(* CODESYS project IndraLogic.project

Project tree, tasks and I/O mapping:
  Sortierstrecke_SPS : IndraControl XM2, Bosch Rexroth AG, order no. dependent on customer specific configuration, version 14.20.34.0
    application Application
      libraries: CommonDataTypes, 3.5.8.40 (OSB AG)
      task PlcTask (cyclic, interval 10 ms, priority 5, watchdog 10 ms x 2) calls PlcProg
      controller/
        function block ColorSensor [ST]: toInt
        function block Compressor [ST]: isActive, start, stop
        function block Conveyor [ST]: isActive, start, stop
        function block Cylinder [ST]: isHome, isWork, moveHome, moveWork
      GVL/
        global variables GVL_IO
        global variables GVL_MasterSlave
        global variables NVL_I_Sorter
        declarations NVL_O_Sorter
      SPS_Communication/
        function block ReadOutputs [ST]: get
        function block SendInputs [ST]: set
      global variables UserVarGlobal
      function CheckBounds [ST]
      program PlcProg [ST]
      program PlcStudentProg [ST]
      Symbols
      visualisation Visualization
    S20_I_O : S20_I_O, Bosch Rexroth AG, version 14.20.10.0
      S20_DIDO_8_1 : S20-DIDO-8/1, Bosch Rexroth AG, order no. R911173745, version Revision=16#0
          settings: Digital Input.IDN = 16#010005DF; Digital Output.IDN = 16#010005DE; Digital Input.IDN = 16#010005DF; Digital Input.Process data out.IDN = 16#00000000; Digital Input.Process data in.IDN = 16#010905DF; Digital Input.Diag out.IDN = 16#00000000; Digital Input.Diag in.IDN = 16#00000000; Digital Input.Io monitoring.IDN_IN = 16#00000000; Digital Input.Io monitoring.IDN_OUT = 16#00000000; Digital Output.IDN = 16#010005DE; Digital Output.Process data out.IDN = 16#010505DE; Digital Output.Process data in.IDN = 16#00000000; Digital Output.Diag out.IDN = 16#00000000; Digital Output.Diag in.IDN = 16#00000000; Digital Output.Io monitoring.IDN_IN = 16#00000000; Digital Output.Io monitoring.IDN_OUT = 16#00000000; PropritaryParameterSet_S-0-1503.0.20.IDN = 16#011405DF; PropritaryParameterSet_S-0-1502.0.2.IDN = 16#010205DE
          output Application.GVL_IO.DO_MotorBeltForward : BOOL  // Digital Output.02
          output Application.GVL_IO.DO_Compressor : BOOL  // Digital Output.03
          output Application.GVL_IO.DO_ValceEjectorOne : BOOL  // Digital Output.12
          output Application.GVL_IO.DO_ValceEjectorTwo : BOOL  // Digital Output.13
          output Application.GVL_IO.DO_ValceEjectorThree : BOOL  // Digital Output.22
          input  Application.GVL_IO.DI_LightBarrierInlet : BOOL  // Digital Input.00
          input  Application.GVL_IO.DI_LightBarrierBehindColor : BOOL  // Digital Input.01
          input  Application.GVL_IO.DI_LightBarrierWhite : BOOL  // Digital Input.10
          input  Application.GVL_IO.DI_LightBarrierRed : BOOL  // Digital Input.11
          input  Application.GVL_IO.DI_LightBarrierBlue : BOOL  // Digital Input.20
          input  Application.GVL_IO.DI_PulseCounter : BOOL  // Digital Input.21
          unmapped channels: Digital Output, Digital Input
      S20_AI_4_U : S20-AI-4-U, Bosch Rexroth AG, order no. R911173256, version Revision=16#0
          settings: Analog Input.IDN = 16#010005E1; Analog Input.IDN = 16#010005E1; Analog Input.Process data out.IDN = 16#00000000; Analog Input.Process data in.IDN = 16#010905E1; Analog Input.Diag out.IDN = 16#00000000; Analog Input.Diag in.IDN = 16#00000000; Analog Input.Io monitoring.IDN_IN = 16#00000000; Analog Input.Io monitoring.IDN_OUT = 16#00000000; PropritaryParameterSet_P-1-0128.0.0.IDN = 16#01009080; PropritaryParameterSet_P-1-0128.0.0.Abort if error = False; PropritaryParameterSet_P-1-0128.0.0.Jump to line if error = False; PropritaryParameterSet_P-1-0128.0.0.SercosAttribute = 16#00000000; PropritaryParameterSet_P-1-0128.0.0 = [16#0C,16#00,16#0C,16#00,16#00,16#02,16#00,16#0F,16#00,16#0F,16#00,16#0F,16#00,16#00,16#00,16#00]
          input  Application.GVL_IO.AI_ColorSensor : WORD  // Analog Input.Analog Input 1
          unmapped channels: Analog Input
    Nicht_verwendet_XM_ : Nicht verwendet (XM), Bosch Rexroth AG, version 14.18.0.0
  text list GlobalTextList
*)

// Sortierstrecke_SPS/Application/GVL/GVL_IO
{attribute 'qualified_only'}
VAR_GLOBAL
		
	//Motors
	DO_MotorBeltForward				: BOOL; //Q1 AT	%QX0.0 
	//Pipes
	DO_Compressor					: BOOL; //Q2 AT	%QX0.1 
	DO_ValceEjectorOne				: BOOL; //Q3 AT	%QX0.2 
	DO_ValceEjectorTwo				: BOOL; //Q4 AT	%QX0.3 
	DO_ValceEjectorThree			: BOOL; //Q5 AT	%QX0.4 
	
	//Pulse Counter
	DI_PulseCounter				 	: BOOL; //I1 AT 	%IX0.5 
	//Light Barriers
	DI_LightBarrierInlet			: BOOL; //I2 AT 	%IX0.0 
	DI_LightBarrierBehindColor 		: BOOL; //I3 AT 	%IX0.1 
	DI_LightBarrierWhite			: BOOL; //I5 AT 	%IX0.2 
	DI_LightBarrierRed	 			: BOOL; //I6 AT 	%IX0.3 
	DI_LightBarrierBlue		 		: BOOL; //I7 AT 	%IX0.4 

	//Color Sensor
	AI_ColorSensor					: WORD; //A4 AT 	%IW2   	
END_VAR

// Sortierstrecke_SPS/Application/GVL/GVL_MasterSlave
{attribute 'qualified_only'}
VAR_GLOBAL
	runMaster : BOOL;
	Stop : BOOL;
END_VAR

// Sortierstrecke_SPS/Application/GVL/NVL_I_Sorter
{attribute 'qualified_only'}
VAR_GLOBAL
	
	//
	//INPUTS:
	//
	
	//Pulse Counter
	DI_PulseCounter				 	: BOOL; //I1 AT 	%IX0.5 
	//Light Barriers
	DI_LightBarrierInlet			: BOOL; //I2 AT 	%IX0.0 
	DI_LightBarrierBehindColor 		: BOOL; //I3 AT 	%IX0.1 
	DI_LightBarrierWhite			: BOOL; //I5 AT 	%IX0.2 
	DI_LightBarrierRed	 			: BOOL; //I6 AT 	%IX0.3 
	DI_LightBarrierBlue		 		: BOOL; //I7 AT 	%IX0.4 

	//Color Sensor
	AI_ColorSensor					: WORD; //A4 AT 	%IW2   	

END_VAR

// Sortierstrecke_SPS/Application/GVL/NVL_O_Sorter
//Diese globale Variablenliste wird über das Netzwerk empfangen.
//Sender: Import aus Datei 'C:\Users\tdie\Documents\HTWK_einzeln\Final\GVLs\Sorter_O.gvl'
//Protokoll: UDP

{attribute 'qualified_only'}
VAR_GLOBAL
	//
	//OUTPUTS:
	//
	
	//Motors
	DO_MotorBeltForward				: BOOL; //Q1 AT	%QX0.0 
	//Pipes
	DO_Compressor					: BOOL; //Q2 AT	%QX0.1 
	DO_ValceEjectorOne				: BOOL; //Q3 AT	%QX0.2 
	DO_ValceEjectorTwo				: BOOL; //Q4 AT	%QX0.3 
	DO_ValceEjectorThree			: BOOL; //Q5 AT	%QX0.4 
	
	Stop : BOOL;
	
END_VAR

// Sortierstrecke_SPS/Application/UserVarGlobal
{attribute 'qualified_only'}
VAR_GLOBAL
	// speichert die Farbe als INT - Wert
	colorAsInt 		: INT;
	
	//zählt die steigenden Flanken des Puls - Counters, um die Position des Objektes
	// auf dem Band zu bestimmen
	clock 	: INT;
END_VAR

// Sortierstrecke_SPS/Application/PlcProg
PROGRAM PlcProg
VAR
	reader : ReadOutputs();
	writer : SendInputs();
END_VAR

//---------------------------------------------------------------
//|		-			run the student code				-		|			
//---------------------------------------------------------------
PlcStudentProg();

//---------------------------------------------------------------
//|		-		Communication, do not modify!			-		|			
//---------------------------------------------------------------

writer.set();
reader.get();

END_PROGRAM

// Sortierstrecke_SPS/Application/PlcStudentProg
PROGRAM PlcStudentProg
VAR
	ColorSensorController	: ColorSensor;
	CompressorController	: Compressor;
	ConveyorController		: Conveyor;
	CylinderController		: Cylinder;
END_VAR

//---------------------------------------------------------------
//|		-		activate or deactivate Master			-		|			
//---------------------------------------------------------------

GVL_MasterSlave.runMaster := FALSE;

//---------------------------------------------------------------
//|		-		write your own code here				-		|			
//---------------------------------------------------------------

ColorSensorController(
	LightValue 				:= GVL_IO.AI_ColorSensor,
	clock					:= UserVarGlobal.clock);
UserVarGlobal.colorAsInt 	:= ColorSensorController.colorAsInt;

CompressorController(
	LightBarrierInlet 		:= GVL_IO.DI_LightBarrierInlet,
	LightBarrierWhite 		:= GVL_IO.DI_LightBarrierWhite,
	LightBarrierBlue 		:= GVL_IO.DI_LightBarrierBlue, 
	LightBarrierRed 		:= GVL_IO.DI_LightBarrierRed);
GVL_IO.DO_Compressor 		:= CompressorController.CompressorM;

ConveyorController(
	LightBarrierWhite		:= GVL_IO.DI_LightBarrierWhite,
	LightBarrierRed			:= GVL_IO.DI_LightBarrierRed,
	LightBarrierBlue		:= GVL_IO.DI_LightBarrierBlue,
	LightBarrierInlet		:= GVL_IO.DI_LightBarrierInlet,
	PulseCounter			:= GVL_IO.DI_PulseCounter);
GVL_IO.DO_MotorBeltForward 	:= ConveyorController.MotorBeltForward;
UserVarGlobal.clock		 	:= ConveyorController.clock;

CylinderController(
	colorAsInt 				:= UserVarGlobal.colorAsInt,
	clock		 			:= UserVarGlobal.clock);
GVL_IO.DO_ValceEjectorOne 	:= CylinderController.ValceEjectorOne;
GVL_IO.DO_ValceEjectorTwo 	:= CylinderController.ValceEjectorTwo;
GVL_IO.DO_ValceEjectorThree := CylinderController.ValceEjectorThree;

END_PROGRAM

// Sortierstrecke_SPS/Application/controller/ColorSensor
FUNCTION_BLOCK ColorSensor
VAR_INPUT
	LightValue	: DWORD;
	clock		: INT;
END_VAR
VAR_OUTPUT
	colorAsInt	: INT;
END_VAR
VAR
	
END_VAR

IF clock = 1 THEN
	THIS^.colorAsInt := toInt();
END_IF

METHOD toInt : INT
VAR_INPUT
END_VAR
IF THIS^.LightValue = 0 THEN
	toInt := 0;	//white
ELSIF THIS^.LightValue = 1 THEN
	toInt := 1; //red
ELSIF THIS^.LightValue = 2 THEN
	toInt := 2; //blue
ELSE 
	toInt := 3; //sollte nicht passieren
END_IF;
END_METHOD

END_FUNCTION_BLOCK

// Sortierstrecke_SPS/Application/controller/Compressor
FUNCTION_BLOCK Compressor

VAR_INPUT
	LightBarrierInlet			: BOOL;
	LightBarrierWhite 		 	: BOOL;
	LightBarrierBlue 			: BOOL;
	LightBarrierRed 			: BOOL;
END_VAR
VAR_OUTPUT
	CompressorM					: BOOL;
END_VAR
VAR
	an : F_TRIG;
	aus : F_TRIG;
END_VAR

an(CLK := LightBarrierInlet);
aus(CLK := LightBarrierWhite AND  LightBarrierBlue AND LightBarrierRed);

//Laden
IF an.Q AND NOT isActive() THEN
	start();
END_IF

//Stoppen
IF aus.Q AND isActive() THEN
	stop();
END_IF

METHOD isActive : BOOL
VAR_INPUT
END_VAR
IF THIS^.CompressorM THEN
	isActive := TRUE;
ELSE
	isActive := FALSE;
END_IF
END_METHOD

METHOD start
VAR_INPUT
END_VAR
THIS^.CompressorM := TRUE;
END_METHOD

METHOD stop
VAR_INPUT
END_VAR
THIS^.CompressorM := FALSE;
END_METHOD

END_FUNCTION_BLOCK

// Sortierstrecke_SPS/Application/controller/Conveyor
FUNCTION_BLOCK Conveyor

VAR_INPUT
	LightBarrierInlet	: BOOL;
	LightBarrierRed		: BOOL;
	LightBarrierWhite	: BOOL;
	LightBarrierBlue	: BOOL;
	
	PulseCounter		: BOOL;
END_VAR

VAR_OUTPUT
	MotorBeltForward	: BOOL;
	clock				: INT;
END_VAR

VAR
	an 					: F_TRIG;
	aus					: F_TRIG;
	PulseTrigger 		: R_TRIG;
END_VAR

an(CLK := LightBarrierInlet);
aus(CLK := LightBarrierRed And LightBarrierWhite And LightBarrierBlue);
//Anschalten 
IF an.Q AND NOT isActive() THEN
	start();
END_IF

//Ausschalten
IF aus.Q THEN
	stop();
END_IF

//Erhöhung der Zeit/Position auf dem Band
PulseTrigger(CLK := PulseCounter);
IF isActive() THEN
	IF PulseTrigger.Q THEN
		clock := clock + 1; 
	END_IF
ELSE
	clock :=0;
END_IF

METHOD isActive : BOOL
VAR_INPUT
END_VAR
IF THIS^.MotorBeltForward THEN
	isActive := TRUE;
ELSE
	isActive := FALSE;
END_IF;
END_METHOD

METHOD start 
VAR_INPUT
END_VAR
THIS^.MotorBeltForward := True;
END_METHOD

METHOD stop
VAR_INPUT
END_VAR
THIS^.MotorBeltForward := FALSE;
END_METHOD

END_FUNCTION_BLOCK

// Sortierstrecke_SPS/Application/controller/Cylinder
FUNCTION_BLOCK Cylinder

VAR_INPUT
	colorAsInt					: INT;
	clock						: INT;
END_VAR

VAR_OUTPUT
	ValceEjectorOne				: BOOL;
	ValceEjectorTwo 			: BOOL;
	ValceEjectorThree			: BOOL;
END_VAR

VAR
END_VAR

IF colorAsInt = 0 AND clock = 2 THEN
	IF isHome(ValceEjectorOne) THEN 
		ValceEjectorOne := moveWork();
	ELSIF isWork(ValceEjectorOne) THEN
		ValceEjectorOne := moveHome();
	END_IF
ELSIF colorAsInt = 1 AND clock = 4 THEN
	IF isHome(ValceEjectorTwo) THEN 
		ValceEjectorTwo := moveWork();
	ELSIF isWork(ValceEjectorTwo) THEN
		ValceEjectorTwo  := moveHome();
	END_IF
ELSIF colorAsInt = 2 AND clock = 6 THEN
	IF isHome(ValceEjectorThree) THEN 
		ValceEjectorThree := moveWork();
	ELSIF isWork(ValceEjectorThree) THEN
		ValceEjectorThree := moveHome();
	END_IF
END_IF

METHOD isHome : BOOL
VAR_INPUT
	cylinder : BOOL;
END_VAR
IF cylinder THEN
	isHome := FALSE;
ELSE
	isHome := TRUE;
END_IF
END_METHOD

METHOD isWork : BOOL
VAR_INPUT
	cylinder : BOOL;
END_VAR
IF cylinder THEN
	isWork := TRUE;
ELSE
	isWork := FALSE;
END_IF
END_METHOD

METHOD moveHome : BOOL
VAR_INPUT
END_VAR
moveHome := False;
END_METHOD

METHOD moveWork : BOOL
VAR_INPUT
END_VAR
moveWork := True;
END_METHOD

END_FUNCTION_BLOCK

// Sortierstrecke_SPS/Application/SPS_Communication/ReadOutputs
FUNCTION_BLOCK ReadOutputs
VAR_INPUT
END_VAR
VAR_OUTPUT
END_VAR
VAR
END_VAR

METHOD get
VAR_INPUT
END_VAR

VAR
	GVL_O_Sorter: INT;
	DO_Compressor: INT;
END_VAR
IF(NOT GVL_MasterSlave.Stop)THEN
	GVL_MasterSlave.Stop := NVL_O_Sorter.Stop;
	IF(GVL_MasterSlave.runMaster)THEN
		GVL_IO.DO_Compressor := NVL_O_Sorter.DO_Compressor;
		GVL_IO.DO_MotorBeltForward := NVL_O_Sorter.DO_MotorBeltForward;
		GVL_IO.DO_ValceEjectorOne := NVL_O_Sorter.DO_ValceEjectorOne;
		GVL_IO.DO_ValceEjectorThree := NVL_O_Sorter.DO_ValceEjectorThree;
		GVL_IO.DO_ValceEjectorTwo := NVL_O_Sorter.DO_ValceEjectorTwo;
	END_IF
ELSE	
	//emergency stop active, set all outputs to false
	GVL_IO.DO_Compressor := FALSE;
	GVL_IO.DO_MotorBeltForward := FALSE;
	GVL_IO.DO_ValceEjectorOne := FALSE;
	GVL_IO.DO_ValceEjectorThree := FALSE;
	GVL_IO.DO_ValceEjectorTwo := FALSE;
END_IF
END_METHOD

END_FUNCTION_BLOCK

// Sortierstrecke_SPS/Application/SPS_Communication/SendInputs
FUNCTION_BLOCK SendInputs
VAR_INPUT
END_VAR
VAR_OUTPUT
END_VAR
VAR
END_VAR

METHOD set
VAR_INPUT
END_VAR
VAR
	GVL_I_Sorter: INT;
END_VAR
NVL_I_Sorter.AI_ColorSensor := GVL_IO.AI_ColorSensor;
NVL_I_Sorter.DI_LightBarrierBehindColor := GVL_IO.DI_LightBarrierBehindColor;
NVL_I_Sorter.DI_LightBarrierBlue := GVL_IO.DI_LightBarrierBlue;
NVL_I_Sorter.DI_LightBarrierInlet := GVL_IO.DI_LightBarrierInlet;
NVL_I_Sorter.DI_LightBarrierRed := GVL_IO.DI_LightBarrierRed;
NVL_I_Sorter.DI_LightBarrierWhite := GVL_IO.DI_LightBarrierWhite;
NVL_I_Sorter.DI_PulseCounter := GVL_IO.DI_PulseCounter;
END_METHOD

END_FUNCTION_BLOCK

// Sortierstrecke_SPS/Application/CheckBounds
(*
General Header
----------------------------------------------------------------------------------------------
Short description      : Function to check access to array within valid bounds.
                         After inserting/removing this function, no online-change will be possible! A complete download will be necessary!
Version                : 14.1.0.0
Author                 : DC-IA/EAM3 (MD)
Date                   : 2015-01-12
Company                : Bosch Rexroth AG
Target                 : IndraLogic XLC/MLC
Functional description : This function will be called implicitly before the read/write access
                         to arrays takes places.
                         The index of the subsequent array accesses is checked for valid
                         limits.
                         In case of invalid access, an error is entered in the diagnostic
                         logbook and the application is stopped due to an access violation to
                         avoid machine damage.
                         In this case, check the callstack (menu Debug/Callstack) and modify
                         the faulty logic. 
Handling specials      : This function increases the cycle time of all IEC-tasks using array
                         accesses. 
                         The increase depends on the number of the read/write accesses to
                         arrays.
                         After inserting/removing this function, no online-change will be possible! 
                         A complete download will be necessary!
						 This is an exemplary implementation of the function. 
                         The implementation has to be adjusted to your application/machine.
						 Per default, the PLC-Task will generate an access violation which leads to
                         an application stop and a F5-error with error reaction respectively.
                         Please verify whether this default behaviour can damage your machine 
                         or lead to a complex recommissioning. 
                         In this case, adapt the error reaction to your application.
						 
                         If your application isn't too time-critical, you should leave this function 
						 while commissioning the machine and production in your application.  
                         If you remove this funciton, ensure that your code is faultless.
                         
                         Do not modify the declaration of this function! 
                         Do not change the attributes above the function header!
----------------------------------------------------------------------------------------------
*)
{attribute 'check_bounds'}
{attribute 'no_check'}
{attribute 'signature_flag' := '1073741824'}
FUNCTION CheckBounds : DINT
VAR_INPUT
	index, lower, upper: DINT;
END_VAR
VAR
	{attribute 'hide'}
	bByte: BYTE;
	ptNull: POINTER TO BYTE :=0;
	errstr: STRING;
	
END_VAR

(*************************************************************
This function was generated by the 'check array access'
option of the controllers 'properties' dialog box.
If you delete this comment, the 'check array access' option
of the controllers 'properties' dialog box will be removed.
**************************************************************)
    (**************************************************************************************************)
    (* The implementation has to be adjusted to your application/machine.                             *)
    (* This is an exemplary implementation of the function.                                           *)
    (* Per default, an access violation is generated to avoid machine damage                          *)
    (* Check the Call Stack (menu Debug/Callstack) and modify the faulty logic!                       *)
    (**************************************************************************************************)

IF  index < lower THEN 
	errstr:= 'CheckBounds: Lower arrayindex ';
	errstr:=CONCAT(STR1:=errstr  , STR2:= DINT_TO_STRING(lower));
	errstr:=CONCAT(STR1:=errstr  , STR2:= ' underrunned by ');
	errstr:=CONCAT(STR1:=errstr  , STR2:= DINT_TO_STRING(index));
//  This pragma may be removed: 
	{info 'CheckBounds: Please implement your own error reaction below'}
//  EXAMPLE 1 (default): 
//  Set a F0-Error into the diagnostic- and error memory
//  Triggering an access violation --> Application will be stopped and leads to a F5-Error

  ML_SetDiagEntry(
	Severity:= E_LOG_SEVERITY.ERROR, 
	Class:= E_LOG_CLASS.CLASS_0, 
	Facility:= E_LOG_FACILITY.USER, 
	Code:= 0, 
	Text:= ADR(errstr));

	bByte:=ptNull^;(*triggering an access violation *)

// EXAMPLE 2:
// Limit the faulty index to the lower index 
//     -> no memory will be overwritten
//     -> Keep PLC-task and motion running
// Set a E0-Warning into the diagnostic- and error memory
// NOTE: There is still an implementation error in your application code!

//  ML_SetDiagEntry(
//	Severity:= E_LOG_SEVERITY.WARNING, 
//	Class:= E_LOG_CLASS.CLASS_0, 
//	Facility:= E_LOG_FACILITY.USER, 
//	Code:= 0, 
//	Text:= ADR(errstr));
// 
//	CheckBounds := lower; //access to the lower index only 
//  return;
	
ELSIF  index > upper THEN
	errstr:= 'CheckBounds: Higher arrayindex ';
	errstr:=CONCAT(STR1:=errstr  , STR2:= DINT_TO_STRING(upper));
	errstr:=CONCAT(STR1:=errstr  , STR2:= ' overrunned by ');
	errstr:=CONCAT(STR1:=errstr  , STR2:= DINT_TO_STRING(index));

//  this pragma may be removed: 
	{info 'CheckBounds: Please implement your own error reaction below'}
//  example 1 (default): 
//  set a F0-Error into the diagnostic- and error memory
//  triggering an access violation --> Application will be stopped and leads to a F5-Error

  ML_SetDiagEntry(
	Severity:= E_LOG_SEVERITY.ERROR, 
	Class:= E_LOG_CLASS.CLASS_0, 
	Facility:= E_LOG_FACILITY.USER, 
	Code:= 0, 
	Text:= ADR(errstr));

	bByte:=ptNull^;(*triggering an access violation *)

//example 2:
// Limit the faulty index to the upper index 
//     -> no memory will be overwritten
//     -> Keep PLC-task and motion running
// Set a E0-Warning into the diagnostic- and error memory
// NOTE: There is still an implementation error in your application code!

//  ML_SetDiagEntry(
//	Severity:= E_LOG_SEVERITY.WARNING, 
//	Class:= E_LOG_CLASS.CLASS_0, 
//	Facility:= E_LOG_FACILITY.USER, 
//	Code:= 0, 
//	Text:= ADR(errstr));
// 
//	CheckBounds := upper; //access to the upper index only 
//  return;

ELSE // access to array is ok  
	CheckBounds := index;
END_IF

END_FUNCTION

// Sortierstrecke_SPS/Application/Visualization
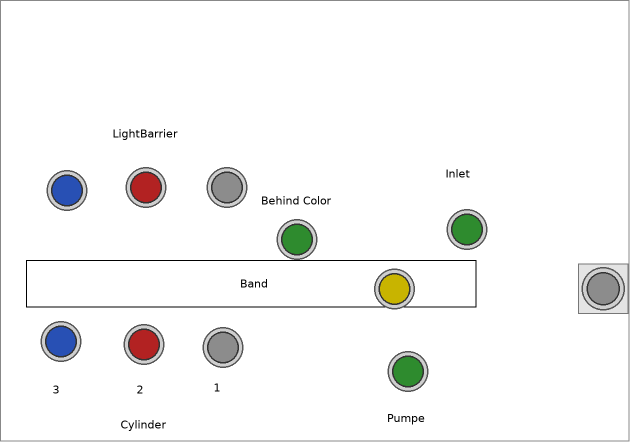
VISUALIZATION Visualization  // 630x442
    Rectangle (26,260 450x47)
    Label (179,269 150x30), "Band"
    Lamp1 (43,167 48x47), variable: GVL_IO.DI_LightBarrierBlue, style: Lamp-Lamp1-Blue
    Lamp1 (122,164 48x47), variable: GVL_IO.DI_LightBarrierRed, style: Lamp-Lamp1-Red
    Lamp1 (203,164 48x47), variable: GVL_IO.DI_LightBarrierWhite, style: Lamp-Lamp1-Gray
    Lamp1 (37,318 48x47), variable: GVL_IO.DO_ValceEjectorThree, style: Lamp-Lamp1-Blue
    Lamp1 (120,321 48x47), variable: GVL_IO.DO_ValceEjectorTwo, style: Lamp-Lamp1-Red
    Lamp1 (199,324 48x47), variable: GVL_IO.DO_ValceEjectorOne, style: Lamp-Lamp1-Gray
    Lamp1 (273,216 48x47), variable: GVL_IO.DI_LightBarrierBehindColor, style: Lamp-Lamp1-Green
    Lamp1 (443,206 48x47), variable: GVL_IO.DI_LightBarrierInlet, style: Lamp-Lamp1-Green
    Lamp1 (384,348 48x47), variable: GVL_IO.DO_Compressor, style: Lamp-Lamp1-Green
    Label (34,410 219x30), "Cylinder"
    Label (24,379 64x22), "3"
    Label (65,375 150x30), "2"
    Label (142,373 150x30), "1"
    Label (380,402 52x33), "Pumpe"
    Label (383,159 150x30), "Inlet"
    Label (221,186 150x30), "Behind Color"
    Label (70,119 150x30), "LightBarrier"
    Lamp1 (371,261 47x56), variable: GVL_IO.DO_MotorBeltForward, style: Lamp-Lamp1-Yellow
    PushSwitch (578,259 50x59), variable: GVL_IO.DI_PulseCounter, behaviour: TOGGLE, style: Switch-PushSwitch-Gray
END_VISUALIZATION
